// TIA Portal V20 export
DATA_BLOCK "DB_FormatMsg"   // DB18
{ S7_Optimized_Access := 'TRUE' }
// stored: MemoryReserve 100
   VAR
      Msg : Array[0..863] of "UDT_FormatMsg";
   END_VAR
BEGIN
END_DATA_BLOCK
